// TIA Portal V18 export
// export: Created 2026-06-09T02:47:52.8345134Z, ExportSetting WithDefaults, DisplayName Totally Integrated Automation Portal, DisplayVersion V18, DisplayName TIA Portal Openness, DisplayVersion V18, DisplayName TIA Portal Version Control Interface, DisplayVersion V18, DisplayName STEP 7 Professional, DisplayVersion V18, DisplayName STEP 7 Safety, DisplayVersion V18, DisplayName WinCC Professional, DisplayVersion V18
DATA_BLOCK "Nalewarka_DB"   // DB3
VERSION : 0.1
// stored: AutoNumber true, DBAccessibleFromOPCUA true, DBAccessibleFromWebserver true, InstanceOfName Nalewarka, InstanceOfType FB
"Nalewarka"
   // VAR
   //    czas_nalewarka : Time;
   // END_VAR
BEGIN
END_DATA_BLOCK
